TYPE SensorOutput :
STRUCT
	SensorName : STRING;
	SensorActive : BOOL;
	
	OutputType : STRING;
	OutputDescription : STRING;
	//OutputINT : INT;
	OutputBOOL : BOOL;
	//OutputREAL : REAL;
END_STRUCT
END_TYPE

(* stored: Version 1.1.0.1, ProductVersion 3.1.4024.9
   DUT SensorOutput: Id {f9187885-03c2-4b52-ac68-929d92f417a0} *)
